FUNCTION_BLOCK NullComponent EXTENDS Component
VAR
END_VAR

END_FUNCTION_BLOCK

(* stored: Version 1.1.0.1, ProductVersion 3.1.4026.18
   POU NullComponent: Id {f1488b7e-691f-4cf3-84f5-5f81b0dae446}, SpecialFunc None *)
